PROGRAM MAIN
VAR
END_VAR

END_PROGRAM

(* stored: Version 1.1.0.1
   POU MAIN: Id {92cb4d8b-5cf4-43e7-bd6a-9944b47a9a9d} *)
